(* IEC 61131-3 sources: AXOpen/src/timers/test, 2 files *)

(* ---- OffDelayTests.st ---- *)
USING AxUnit;
USING AXOpen.Timers;
USING AXOpen.Rtc;
USING AXOpen.Logging;
USING AXOpen.Core;
USING AXOpen.Rtc;

NAMESPACE AXOpen.Timers_tests

    {TestFixture}
    CLASS AxoOffDelayTimersTests
        VAR PROTECTED
            _context : TestContext;
            _inspectedBool : BOOL;
            _rtcMock :  AxoRtcMock;
            _signal : BOOL;
            _testTimerOnDelay: AXOpen.Timers.OnDelayContext;
            _testTimerOffDelay: AXOpen.Timers.OffDelayContext;
            _testTimeDelay: LTIME := LTIME#5s;
        END_VAR

        METHOD PRIVATE Initialize
            _context.InjectRtc(_rtcMock);
        END_METHOD

        {Test}
        METHOD PUBLIC Timer_offDelay_class_output_test
            THIS.Initialize();

            _context.Open();

            _rtcMock.SetNowUTC(LDT#1980-01-23-13:14:33.123456);
            _signal := TRUE;
            _testTimerOffDelay.OffDelay(_context, _signal, _testTimeDelay);
            Assert.Equal(TRUE, _testTimerOffDelay.output);

            //move 6 seconds in future, timer stil don't count, true is output
            _rtcMock.SetNowUTC(LDT#1980-01-23-13:14:39.123456);
            _testTimerOffDelay.OffDelay(_context, _signal, _testTimeDelay);
            Assert.Equal(TRUE, _testTimerOffDelay.output);

            //here, timer starts count
            _rtcMock.SetNowUTC(LDT#1980-01-23-13:14:41.123456);
            _signal := FALSE;
            _testTimerOffDelay.OffDelay(_context, _signal, _testTimeDelay);
            Assert.Equal(TRUE, _testTimerOffDelay.output);

            //here, timer should hit delay and turn off signal
            _rtcMock.SetNowUTC(LDT#1980-01-23-13:14:46.123456);
            _testTimerOffDelay.OffDelay(_context, _signal, _testTimeDelay);
            Assert.Equal(FALSE, _testTimerOffDelay.output);

            _context.Close();
        END_METHOD

        {Test}
        METHOD PUBLIC Timer_offDelay_overall_test
            THIS.Initialize();

            _context.Open();

            //all turn off, previous signal was false, input is false, output should be false
            _rtcMock.SetNowUTC(LDT#1980-01-23-13:14:30.0);
            _signal := FALSE;
            _testTimerOffDelay.OffDelay(_context, _signal, _testTimeDelay);
            Assert.Equal(FALSE, _testTimerOffDelay.output);

            //after 1 second, turn on signal, output should be on
            _rtcMock.SetNowUTC(LDT#1980-01-23-13:14:31.0);
            _signal := TRUE;
            _testTimerOffDelay.OffDelay(_context, _signal, _testTimeDelay);
            Assert.Equal(TRUE, _testTimerOffDelay.output);

            //after 2 second, turn off signal, FALLING EDGE detected, output should be on, timer should start counting
            _rtcMock.SetNowUTC(LDT#1980-01-23-13:14:32.0);
            _signal := FALSE;
            _testTimerOffDelay.OffDelay(_context, _signal, _testTimeDelay);
            Assert.Equal(TRUE, _testTimerOffDelay.output);

            //after 7 second, timer count passed delay, output should be false
            _rtcMock.SetNowUTC(LDT#1980-01-23-13:14:35.0);
            _testTimerOffDelay.OffDelay(_context, _signal, _testTimeDelay);
            Assert.Equal(FALSE, _testTimerOffDelay.output);

            //after 10 second, rising edge was detected, timer is reseted and output should be true
            _rtcMock.SetNowUTC(LDT#1980-01-23-13:14:40.0);
            _signal := TRUE;
            _testTimerOffDelay.OffDelay(_context, _signal, _testTimeDelay);
            Assert.Equal(TRUE, _testTimerOffDelay.output);

            //after 11 second, falling edge was detected, timer should start count again
            _rtcMock.SetNowUTC(LDT#1980-01-23-13:14:41.0);
            _signal := FALSE;
           _testTimerOffDelay.OffDelay(_context, _signal, _testTimeDelay);
            Assert.Equal(TRUE, _testTimerOffDelay.output);

            //after 13 second, rising edge was detected, timer is reseted, output is still true
            _rtcMock.SetNowUTC(LDT#1980-01-23-13:14:43.0);
            _signal := TRUE;
            _testTimerOffDelay.OffDelay(_context, _signal, _testTimeDelay);
            Assert.Equal(TRUE, _testTimerOffDelay.output);

            _context.Close();
        END_METHOD

        {Test}
        METHOD PUBLIC Timer_offDelay_method_output_test
            VAR_TEMP
                _methodOutput: BOOL;
            END_VAR
            THIS.Initialize();

            _context.Open();

            _rtcMock.SetNowUTC(LDT#1980-01-23-13:14:33.123456);
            _signal := TRUE;
            _methodOutput := _testTimerOffDelay.OffDelay(_context, _signal, _testTimeDelay);
            Assert.Equal(TRUE, _methodOutput);

            //move 6 seconds in future, timer stil don't count, true is output
            _rtcMock.SetNowUTC(LDT#1980-01-23-13:14:39.123456);
            _methodOutput := _testTimerOffDelay.OffDelay(_context, _signal, _testTimeDelay);
            Assert.Equal(TRUE, _methodOutput);

            //here, timer starts count
            _rtcMock.SetNowUTC(LDT#1980-01-23-13:14:41.123456);
            _signal := FALSE;
            _methodOutput := _testTimerOffDelay.OffDelay(_context, _signal, _testTimeDelay);
            Assert.Equal(TRUE, _methodOutput);

            //here, timer should hit delay and turn off signal
            _rtcMock.SetNowUTC(LDT#1980-01-23-13:14:46.123456);
            _methodOutput := _testTimerOffDelay.OffDelay(_context, _signal, _testTimeDelay);
            Assert.Equal(FALSE, _methodOutput);

            _context.Close();
        END_METHOD

        {Test}
        METHOD PUBLIC Timer_offDelay_delay_is_not_reached_output_is_true
            VAR_TEMP
                _methodOutput: BOOL;
            END_VAR
            THIS.Initialize();

            _context.Open();

            _rtcMock.SetNowUTC(LDT#1980-01-23-13:14:33.123456);
            _signal := TRUE;
            _methodOutput := _testTimerOffDelay.OffDelay(_context, _signal, _testTimeDelay);
            Assert.Equal(TRUE, _methodOutput);

            //move 3 seconds in future
            _rtcMock.SetNowUTC(LDT#1980-01-23-13:14:36.123456);
            _methodOutput := _testTimerOffDelay.OffDelay(_context, _signal, _testTimeDelay);
            Assert.Equal(TRUE, _methodOutput);

            _context.Close();
        END_METHOD

        {Test}
        METHOD PUBLIC Timer_offDelay_zero_delay
            VAR_TEMP
                _resultET : BOOL;
            END_VAR
            THIS.Initialize();

            //arange
            _context.Open();
            _testTimeDelay := LT#0s;
            _rtcMock.SetNowUTC(LDT#1980-01-23-13:14:33.123456);
            _signal := TRUE;

            //act/assert
            _testTimerOffDelay.OffDelay(_context, _signal, _testTimeDelay);
            Assert.Equal(TRUE, _testTimerOffDelay.output);

            _context.Close();
        END_METHOD

        {Test}
        METHOD PUBLIC Timer_offDelay_evertyhing_off
            VAR_TEMP
                _resultET : BOOL;
            END_VAR
            THIS.Initialize();

            //arange
            _context.Open();

            _rtcMock.SetNowUTC(LDT#1980-01-23-13:14:33.123456);
            _signal := FALSE;

            //act/assert
            _testTimerOffDelay.OffDelay(_context, _signal, _testTimeDelay);
            Assert.Equal(FALSE, _testTimerOffDelay.output);

            _context.Close();
        END_METHOD

       END_CLASS
END_NAMESPACE

(* ---- test.st ---- *)
USING AXOpen.Timers;
USING AXOpen.Rtc;
USING AXOpen.Logging;
USING AXOpen.Core;
USING AXOpen.Rtc;
USING AxUnit;

NAMESPACE AXOpen.Timers_tests

    CLASS PUBLIC _NULL_LOGGER IMPLEMENTS IAxoLogger
        METHOD PUBLIC Log
            VAR_INPUT
                _message : STRING[80];
                _level : eLogLevel;
                _sender : IAxoObject;
            END_VAR
            ;
        END_METHOD

        METHOD PUBLIC Log
            VAR_INPUT
                _message : STRING[80];
                _level : eLogLevel;
            END_VAR
            ;
        END_METHOD

        METHOD PUBLIC SetMinimumLevel : IAxoLoggerConfig
            VAR_INPUT
                _level : eLogLevel;
            END_VAR
            ;
        END_METHOD
    END_CLASS

    CLASS AxoRtcMock IMPLEMENTS IAxoRtc
        VAR PRIVATE
            _NowUTC : LDATE_AND_TIME;
        END_VAR

        METHOD INTERNAL SetNowUTC : LDATE_AND_TIME
            VAR_INPUT
                Set :  LDATE_AND_TIME;
            END_VAR;
            _NowUTC := Set;
        END_METHOD

        METHOD PUBLIC NowUTC : LDATE_AND_TIME
            NowUTC := _NowUTC;
        END_METHOD
    END_CLASS

    CLASS TestContext IMPLEMENTS IAxoContext
        VAR PROTECTED
            _openCounter : ULINT;
            _closeCounter : ULINT;
            _identityCounter : ULINT;
            _rtc :  IAxoRtc;
         END_VAR
        METHOD PUBLIC Open : ULINT
            _openCounter := _openCounter + ULINT#1;
        END_METHOD

        METHOD PUBLIC Close : ULINT
            _closeCounter := _closeCounter + ULINT#1;
        END_METHOD

        METHOD PUBLIC OpenCycleCount : ULINT
            OpenCycleCount := _openCounter;
        END_METHOD

        METHOD PUBLIC ClosedCycleCount : ULINT
            ClosedCycleCount := _closeCounter;
        END_METHOD

        METHOD PUBLIC CreateIdentity : ULINT
            _identityCounter := _identityCounter + ULINT#1;
            CreateIdentity := _identityCounter;
        END_METHOD

        METHOD PUBLIC GetRtc : IAxoRtc ;
            GetRtc := _rtc;
        END_METHOD

        METHOD PUBLIC InjectRtc
             VAR_INPUT Rtc : IAxoRtc;
            END_VAR ;

            _rtc := Rtc;
        END_METHOD

        VAR PRIVATE
            NULL_LOGGER : _NULL_LOGGER;
        END_VAR
        METHOD PUBLIC GetLogger : AXOpen.Logging.IAxoLogger GetLogger := NULL_LOGGER; END_METHOD
        METHOD PUBLIC InjectLogger VAR_INPUT _logger : AXOpen.Logging.IAxoLogger; END_VAR ; END_METHOD

    END_CLASS

    {TestFixture}
    CLASS AxoTimersTests
        VAR PROTECTED
            _context : TestContext;
            _inspectedBool : BOOL;
            _rtcMock :  AxoRtcMock;
            _signal : BOOL;
            _testTimer: AXOpen.Timers.OnDelayContext;
            _testTimeDelay: LTIME;
        END_VAR

        METHOD PRIVATE Initialize
            _context.InjectRtc(_rtcMock);
            //_sequencer.Initialize(_context);
        END_METHOD

        {Test}
        METHOD PUBLIC Timer_test_pass
            THIS.Initialize();

            _context.Open();

            _rtcMock.SetNowUTC(LDT#1980-01-23-13:14:33.123456);
            _signal := TRUE;
            _testTimeDelay := LTIME#5s;

            _testTimer.OnDelay(_context, _signal, _testTimeDelay);

            Assert.Equal(FALSE, _testTimer.output);

            //move 6 seconds in future
            _rtcMock.SetNowUTC(LDT#1980-01-23-13:14:39.123456);

            _testTimer.OnDelay(_context, _signal, _testTimeDelay);

            Assert.Equal(TRUE, _testTimer.output);

            //move 8 seconds in future
            _rtcMock.SetNowUTC(LDT#1980-01-23-13:14:41.123456);

            _signal := FALSE;

            _testTimer.OnDelay(_context, _signal, _testTimeDelay);

            Assert.Equal(FALSE, _testTimer.output);

            //_testBool := _digitalInspector.Inspect(_sequencer,_inspectedBool).Done();
            //_digitalInspector.WithCoordinator(_sequencer).Inspect(_sequencer,_inspectedBool).OnFail().CarryOn();

        // WHILE NOT  _digitalInspector.Inspect(_sequencer,_inspectedBool).Done() DO
        //         ;
        //     END_WHILE;

           // Assert.Equal(eInspectorResult#Passed, _digitalInspector.Data()^.Result);

            _context.Close();
        END_METHOD

        // {Test}
        // METHOD PUBLIC Inspection_should_pass
        //     THIS.Initialize();

        //     _context.Open();
        //     _sequencer.Invoke();
        //     _sequencer.Open();

        //     _rtcMock.SetNowUTC(LDT#1980-01-23-13:14:33.123456);
        //     _inspectedBool := TRUE;
        //     _digitalInspector.Data()^.RequiredStatus := TRUE;

        //     _testBool := _digitalInspector.Inspect(_sequencer,_inspectedBool).Done();

        //     _rtcMock.SetNowUTC(LDT#1980-01-23-13:14:38.123456);

        //     _testBool := _digitalInspector.Inspect(_sequencer,_inspectedBool).Done();
        //     //_digitalInspector.WithCoordinator(_sequencer).Inspect(_sequencer,_inspectedBool).OnFail().CarryOn();

        // // WHILE NOT  _digitalInspector.Inspect(_sequencer,_inspectedBool).Done() DO
        // //         ;
        // //     END_WHILE;

        //     Assert.Equal(eInspectorResult#Passed, _digitalInspector.Data()^.Result);

        //     _context.Close();
        // END_METHOD

        // {Test}
        // METHOD PUBLIC Inspection_is_bypassed
        //     THIS.Initialize();
        //     _context.Open();
        //     _sequencer.Invoke();
        //     _sequencer.Open();

        //     _inspectedBool := FALSE;
        //     _digitalInspector.Data()^.RequiredStatus := TRUE;
        //     _digitalInspector.Data()^.IsByPassed := TRUE;

        //     _digitalInspector.Inspect(_sequencer,_inspectedBool);

        //     // // WHILE NOT  DO
        //     // //     ;
        //     // // END_WHILE;

        //    Assert.Equal(eInspectorResult#Bypassed, _digitalInspector.Data()^.Result);
        //     // // ELSE
        //     // //     Assert.Equal(eInspectorResult#Running, _digitalInspector.Data()^.Result);

        //     _context.Close();
        //     ;
        // END_METHOD

        // {Test}
        // METHOD PUBLIC Execute_should_not_crush_when_coordinator_not_passed
        //     _stepOne.Execute(coord := NULL);
        // END_METHOD

       END_CLASS
END_NAMESPACE
